// TIA Portal V20 export
DATA_BLOCK "RealDbName"   // DB7
   VAR RETAIN
      IO { S7_SetPoint := 'True'} : "TypeDOL";
   END_VAR
BEGIN
   IO.InHand := FALSE;
   IO.Running := FALSE;
END_DATA_BLOCK
